TYPE ST_PhasesCommon :
STRUCT
  L1_L2_V : REAL;
END_STRUCT
END_TYPE

(* stored: Version 1.1.0.1, ProductVersion 3.1.4024.12
   DUT ST_PhasesCommon: Id {6a70baa2-afbe-4282-b59d-eaebeb4421f6} *)
